{attribute 'qualified_only'}
{attribute 'strict'}
TYPE GridPointType :
(
	normal := 0,
	stationLeft,
	stationRight,
	stationApproachLeft,
	stationApproachRight,
	charger,
	waitingSpot
);
END_TYPE

(* stored: Version 1.1.0.1, ProductVersion 3.1.4024.11
   DUT GridPointType: Id {577ef664-3e83-4697-9fe7-2af0ee924810} *)
